(* IEC 61131-3 sources: volt/packages/volt-lsp-iec/test-corpus/CodesysTestProject/Device/Plc Logic/Application/Library Manager/CmpApp, 69 files *)

(* ---- APP_MEMORY_SEGMENT.dut ---- *)
TYPE APP_MEMORY_SEGMENT :
STRUCT
	WTYPE : WORD;
	WAREA : WORD;
	DWOFFSET : DWORD;
	DWSIZE : DWORD;
	DWHIGHESTUSEDADDRESS : DWORD;
END_STRUCT
END_TYPE

(* ---- APPLICATION.dut ---- *)
TYPE APPLICATION :
STRUCT
	PAPPPARENT : POINTER TO APPLICATION;
	IID : UDINT;
	CODEGUID : ARRAY [0..15] OF BYTE;
	DATAGUID : ARRAY [0..15] OF BYTE;
	UDISTATE : UDINT;
	UDIOPSTATE : UDINT;
	HBOOTPROJECT : RTS_IEC_HANDLE;
	HDEBUGTASK : RTS_IEC_HANDLE;
	PFGLOBALINIT : POINTER TO BYTE;
	PFGLOBALEXIT : POINTER TO BYTE;
	HSESSIONIDPOOL : RTS_IEC_HANDLE;
	HFORCEPOOL : RTS_IEC_HANDLE;
	HBPPOOL : RTS_IEC_HANDLE;
	BPERSISTENTFORCE : DINT;
	SZNAME : STRING(MAX_LEN_APPLNAME);
	UDIPSVERSION : UDINT;
	UDITARGETSETTINGVERSION : UDINT;
END_STRUCT
END_TYPE

(* ---- APPLICATION_INFO.dut ---- *)
TYPE APPLICATION_INFO :
STRUCT
	PSTPROJECTNAME : POINTER TO STRING(255);
	PSTAUTHOR : POINTER TO STRING(255);
	PSTVERSION : POINTER TO STRING(255);
	PSTDESCRIPTION : POINTER TO STRING(255);
	PSTPROFILE : POINTER TO STRING(255);
	DTLASTCHANGES : DATE_AND_TIME;
END_STRUCT
END_TYPE

(* ---- EVTPARAM_CMPAPP.dut ---- *)
TYPE EVTPARAM_CMPAPP :
STRUCT
	PAPP : POINTER TO APPLICATION;
END_STRUCT
END_TYPE

(* ---- EVTPARAM_CMPAPPALLBOOTAPPSLOADED.dut ---- *)
TYPE EVTPARAM_CMPAPPALLBOOTAPPSLOADED :
STRUCT
	NTOTALBOOTAPPS : DINT;
	NSUCCESSFULLYLOADEDBOOTAPPS : DINT;
END_STRUCT
END_TYPE

(* ---- EVTPARAM_CMPAPPCOMM.dut ---- *)
TYPE EVTPARAM_CMPAPPCOMM :
STRUCT
	PAPP : POINTER TO APPLICATION;
	UDISESSIONID : UDINT;
	UDIAPPSESSIONID : UDINT;
END_STRUCT
END_TYPE

(* ---- EVTPARAM_CMPAPPCOMMCYCLE.dut ---- *)
TYPE EVTPARAM_CMPAPPCOMMCYCLE :
STRUCT
	ULPARAM1 : __XWORD;
	ULPARAM2 : __XWORD;
END_STRUCT
END_TYPE

(* ---- EVTPARAM_CMPAPPCONFIG.dut ---- *)
TYPE EVTPARAM_CMPAPPCONFIG :
STRUCT
	PAPP : POINTER TO APPLICATION;
	PSZCONFIGAPPLICATION : POINTER TO STRING;
END_STRUCT
END_TYPE

(* ---- EVTPARAM_CMPAPPDELETE.dut ---- *)
TYPE EVTPARAM_CMPAPPDELETE :
STRUCT
	PAPP : POINTER TO APPLICATION;
	ULDELETEREASON : UDINT;
END_STRUCT
END_TYPE

(* ---- EVTPARAM_CMPAPPDENY.dut ---- *)
TYPE EVTPARAM_CMPAPPDENY :
STRUCT
	PAPP : POINTER TO APPLICATION;
	UDIDENY : UDINT;
END_STRUCT
END_TYPE

(* ---- EVTPARAM_CMPAPPDENYDELETE.dut ---- *)
TYPE EVTPARAM_CMPAPPDENYDELETE :
STRUCT
	PAPP : POINTER TO APPLICATION;
	UDISHUTDOWN : UDINT;
	UDIDENY : UDINT;
END_STRUCT
END_TYPE

(* ---- EVTPARAM_CMPAPPDENYLOADBOOTPROJECT.dut ---- *)
TYPE EVTPARAM_CMPAPPDENYLOADBOOTPROJECT :
STRUCT
	PSZAPPNAME : POINTER TO STRING;
	BDENY : DINT;
END_STRUCT
END_TYPE

(* ---- EVTPARAM_CMPAPPDENYSTART.dut ---- *)
TYPE EVTPARAM_CMPAPPDENYSTART :
STRUCT
	PAPP : POINTER TO APPLICATION;
	BDENY : DINT;
END_STRUCT
END_TYPE

(* ---- EVTPARAM_CMPAPPDENYSTOP.dut ---- *)
TYPE EVTPARAM_CMPAPPDENYSTOP :
STRUCT
	PAPP : POINTER TO APPLICATION;
	ULSTOPREASON : DWORD;
	BDENY : DINT;
END_STRUCT
END_TYPE

(* ---- EVTPARAM_CMPAPPEXCEPTION.dut ---- *)
TYPE EVTPARAM_CMPAPPEXCEPTION :
STRUCT
	PAPP : POINTER TO APPLICATION;
	HIECTASK : RTS_IEC_HANDLE;
	UDIEXCEPTION : UDINT;
END_STRUCT
END_TYPE

(* ---- EVTPARAM_CMPAPPEXIT.dut ---- *)
TYPE EVTPARAM_CMPAPPEXIT :
STRUCT
	PAPP : POINTER TO APPLICATION;
	ULEXITREASON : UDINT;
END_STRUCT
END_TYPE

(* ---- EVTPARAM_CMPAPPOEMSERVICETAG.dut ---- *)
TYPE EVTPARAM_CMPAPPOEMSERVICETAG :
STRUCT
	PAPP : POINTER TO APPLICATION;
	UDICHANNELID : UDINT;
	UDITOPLEVELTAG : UDINT;
	UDIHEADERTAG : UDINT;
	UDIREADER : UDINT;
	UDIWRITER : UDINT;
	UDIRESULT : UDINT;
END_STRUCT
END_TYPE

(* ---- EVTPARAM_CMPAPPOPERATINGSTATECHANGED.dut ---- *)
TYPE EVTPARAM_CMPAPPOPERATINGSTATECHANGED :
STRUCT
	PAPP : POINTER TO APPLICATION;
	UDIPREVOPSTATE : UDINT;
END_STRUCT
END_TYPE

(* ---- EVTPARAM_CMPAPPPREPARELOADBOOTPROJECT.dut ---- *)
TYPE EVTPARAM_CMPAPPPREPARELOADBOOTPROJECT :
STRUCT
	PSZAPPNAME : POINTER TO STRING;
END_STRUCT
END_TYPE

(* ---- EVTPARAM_CMPAPPREGISTERBOOTPROJECT.dut ---- *)
TYPE EVTPARAM_CMPAPPREGISTERBOOTPROJECT :
STRUCT
	PSZAPPNAME : POINTER TO STRING;
END_STRUCT
END_TYPE

(* ---- EVTPARAM_CMPAPPRESET.dut ---- *)
TYPE EVTPARAM_CMPAPPRESET :
STRUCT
	PAPP : POINTER TO APPLICATION;
	EWRESETOPTION : RESET_OPTION;
END_STRUCT
END_TYPE

(* ---- EVTPARAM_CMPAPPRESETALLAPPLICATIONS.dut ---- *)
TYPE EVTPARAM_CMPAPPRESETALLAPPLICATIONS :
STRUCT
	EWRESETOPTION : RESET_OPTION;
END_STRUCT
END_TYPE

(* ---- EVTPARAM_CMPAPPRETAINBACKUPSTATE.dut ---- *)
TYPE EVTPARAM_CMPAPPRETAINBACKUPSTATE :
STRUCT
	PSZBOOTPROJECTNAME : POINTER TO STRING;
	UIBACKUPSTATE : UINT;
END_STRUCT
END_TYPE

(* ---- EVTPARAM_CMPAPPSOURCEDOWNLOAD.dut ---- *)
TYPE EVTPARAM_CMPAPPSOURCEDOWNLOAD :
STRUCT
	PSZARCHIVENAME : POINTER TO STRING;
	USIBEGIN : USINT;
END_STRUCT
END_TYPE

(* ---- EVTPARAM_CMPAPPSTATECHANGED.dut ---- *)
TYPE EVTPARAM_CMPAPPSTATECHANGED :
STRUCT
	PAPP : POINTER TO APPLICATION;
	UDIPREVSTATE : UDINT;
END_STRUCT
END_TYPE

(* ---- EVTPARAM_CMPAPPSTOP.dut ---- *)
TYPE EVTPARAM_CMPAPPSTOP :
STRUCT
	PAPP : POINTER TO APPLICATION;
	ULSTOPREASON : DWORD;
END_STRUCT
END_TYPE

(* ---- PROJECT_INFO.dut ---- *)
TYPE PROJECT_INFO :
STRUCT
	STPROJECT : STRING;
	STTITLE : STRING;
	STVERSION : STRING;
	STAUTHOR : STRING;
	STDESCRIPTION : STRING;
END_STRUCT
END_TYPE

(* ---- RESET_OPTION.dut ---- *)
TYPE RESET_OPTION :
(
	RTS_RESET := 0,
	RTS_RESET_COLD := 1,
	RTS_RESET_ORIGIN := 2,
	RTS_RESET_ORIGIN_DEVICE := 3
);
END_TYPE

(* ---- APPLICATIONFLAGS.gvl ---- *)
VAR_GLOBAL
	AF_SYSTEM_APPLICATION : UDINT := 16#10000;
	AF_IOCONFIG_BYTE_ADDRESSING : UDINT := 16#20000;
	AF_IOCONFIG_BIT_WORD_ADDRESSING : UDINT := 16#40000;
	AF_KEEP_AT_PARENT_ONLINE_CHANGE : UDINT := 16#80000;
	AF_ALLOW_SYMBOLIC_VARIABLE_ACCESS_IN_SYNC_WITH_IEC_TASK : UDINT := 16#100000;
	AF_SIGNED_APPLICATION : UDINT := 16#200000;
	AF_ENCRYPTED_APPLICATION : UDINT := 16#400000;
	AF_DEVICE_APPLICATION : UDINT := 16#800000;
	AF_APPLICATION_STOP_PARENT_APPS_ON_EXCEPTION : UDINT := 16#1000000;
END_VAR

(* ---- APPLICATIONSTATE.gvl ---- *)
VAR_GLOBAL
	AS_NONE : UDINT := 16#0;
	AS_RUN : UDINT := 16#1;
	AS_STOP : UDINT := 16#2;
	AS_DEBUG_HALT_ON_BP : UDINT := 16#3;
	AS_DEBUG_STEP : UDINT := 16#4;
	AS_SINGLE_CYCLE : UDINT := 16#5;
END_VAR

(* ---- AREATYPES.gvl ---- *)
VAR_GLOBAL
	DA_NONE : UINT := 16#0;
	DA_DATA : UINT := 16#1;
	DA_CONSTANT : UINT := 16#2;
	DA_INPUT : UINT := 16#4;
	DA_OUTPUT : UINT := 16#8;
	DA_MEMORY : UINT := 16#10;
	DA_RETAIN : UINT := 16#20;
	DA_CODE : UINT := 16#40;
	DA_PERSISTENT : UINT := 16#100;
	DA_ALL : UINT := 16#FFFF;
END_VAR

(* ---- EVENTIDS.gvl ---- *)
VAR_GLOBAL
	CMPID_CMPAPP : DWORD := 16#2;
	EVTPARAMID_CMPAPP : WORD := 16#1;
	EVTVERSION_CMPAPP : WORD := 16#1;
	EVTPARAMID_CMPAPPCONFIG : WORD := 16#1;
	EVTVERSION_CMPAPPCONFIG : WORD := 16#1;
	EVTPARAMID_CMPAPPRESET : WORD := 16#1;
	EVTVERSION_CMPAPPRESET : WORD := 16#2;
	EVTPARAMID_CMPAPPSTOP : WORD := 16#2;
	EVTVERSION_CMPAPPSTOP : WORD := 16#1;
	EVTPARAMID_CMPAPPEXIT : WORD := 16#1;
	EVTVERSION_CMPAPPEXIT : WORD := 16#2;
	EVTPARAMID_CMPAPPDELETE : WORD := 16#1;
	EVTVERSION_CMPAPPDELETE : WORD := 16#2;
	EVTPARAMID_CMPAPPDENYSTART : WORD := 16#3;
	EVTVERSION_CMPAPPDENYSTART : WORD := 16#1;
	EVTPARAMID_CMPAPPDENYSTOP : WORD := 16#4;
	EVTVERSION_CMPAPPDENYSTOP : WORD := 16#1;
	EVTPARAMID_CMPAPPALLBOOTAPPSLOADED : WORD := 16#5;
	EVTVERSION_CMPAPPALLBOOTAPPSLOADED : WORD := 16#1;
	EVTPARAMID_CMPAPPDENYLOADBOOTPROJECT : WORD := 16#6;
	EVTVERSION_CMPAPPDENYLOADBOOTPROJECT : WORD := 16#1;
	EVTPARAMID_CMPAPPPREPARELOADBOOTPROJECT : WORD := 16#7;
	EVTVERSION_CMPAPPPREPARELOADBOOTPROJECT : WORD := 16#1;
	EVTPARAMID_CMPAPPEXCEPTION : WORD := 16#8;
	EVTVERSION_CMPAPPEXCEPTION : WORD := 16#1;
	EVTPARAMID_CMPAPPREGISTERBOOTPROJECT : WORD := 16#9;
	EVTVERSION_CMPAPPREGISTERBOOTPROJECT : WORD := 16#1;
	EVTPARAMID_CMPAPPOPERATINGSTATECHANGED : WORD := 16#A;
	EVTVERSION_CMPAPPOPERATINGSTATECHANGED : WORD := 16#1;
	EVTPARAMID_CMPAPPSOURCEDOWNLOAD : WORD := 16#B;
	EVTVERSION_CMPAPPSOURCEDOWNLOAD : WORD := 16#1;
	EVTPARAMID_CMPAPPCOMM : WORD := 16#C;
	EVTVERSION_CMPAPPCOMM : WORD := 16#2;
	EVTPARAMID_CMPAPPDENY : WORD := 16#D;
	EVTVERSION_CMPAPPDENY : WORD := 16#1;
	EVTPARAMID_CMPAPPDENYDELETE : WORD := 16#E;
	EVTVERSION_CMPAPPDENYDELETE : WORD := 16#1;
	EVTPARAMID_CMPAPPOEMSERVICETAG : WORD := 16#F;
	EVTVERSION_CMPAPPOEMSERVICETAG : WORD := 16#1;
	EVTPARAMID_CMPAPPCOMMCYCLE : WORD := 16#17;
	EVTVERSION_CMPAPPCOMMCYCLE : WORD := 16#1;
	EVTPARAMID_CMPAPPSTATECHANGED : WORD := 16#18;
	EVTVERSION_CMPAPPSTATECHANGED : WORD := 16#1;
	EVTPARAMID_CMPAPPRETAINBACKUPSTATE : WORD := 16#1B;
	EVTVERSION_CMPAPPRETAINBACKUPSTATE : WORD := 16#1;
	EVTPARAMID_CMPAPPRESETALLAPPLICATIONS : WORD := 16#1C;
	EVTVERSION_CMPAPPRESETALLAPPLICATIONS : WORD := 16#1;
	APP_STOP_REASON_UNKNOWN : DWORD := 0;
	APP_STOP_REASON_SHUTDOWN : DWORD := 1;
	APP_STOP_REASON_RESET : DWORD := 2;
	APP_STOP_REASON_EXCEPTION : DWORD := 3;
	APP_STOP_REASON_USER : DWORD := 4;
	APP_STOP_REASON_IECPROGRAM : DWORD := 5;
	APP_STOP_REASON_DELETE : DWORD := 6;
	EVT_PREPARESTART : DWORD := (SHL(UINT_TO_DWORD(EventClass.EVTCLASS_INFO), 16) OR 16#1);
	EVT_STARTDONE : DWORD := (SHL(UINT_TO_DWORD(EventClass.EVTCLASS_INFO), 16) OR 16#2);
	EVT_PREPARESTOP : DWORD := (SHL(UINT_TO_DWORD(EventClass.EVTCLASS_INFO), 16) OR 16#3);
	EVT_STOPDONE : DWORD := (SHL(UINT_TO_DWORD(EventClass.EVTCLASS_INFO), 16) OR 16#4);
	EVT_PREPARERESET : DWORD := (SHL(UINT_TO_DWORD(EventClass.EVTCLASS_INFO), 16) OR 16#5);
	EVT_RESETDONE : DWORD := (SHL(UINT_TO_DWORD(EventClass.EVTCLASS_INFO), 16) OR 16#6);
	EVT_PREPAREONLINECHANGE : DWORD := (SHL(UINT_TO_DWORD(EventClass.EVTCLASS_INFO), 16) OR 16#7);
	EVT_ONLINECHANGEDONE : DWORD := (SHL(UINT_TO_DWORD(EventClass.EVTCLASS_INFO), 16) OR 16#8);
	EVT_PREPAREDOWNLOAD : DWORD := (SHL(UINT_TO_DWORD(EventClass.EVTCLASS_INFO), 16) OR 16#9);
	EVT_DOWNLOADDONE : DWORD := (SHL(UINT_TO_DWORD(EventClass.EVTCLASS_INFO), 16) OR 16#A);
	EVT_CODEINITDONE : DWORD := (SHL(UINT_TO_DWORD(EventClass.EVTCLASS_INFO), 16) OR 16#B);
	EVT_PREPAREDELETE : DWORD := (SHL(UINT_TO_DWORD(EventClass.EVTCLASS_INFO), 16) OR 16#C);
	EVT_DELETEDONE : DWORD := (SHL(UINT_TO_DWORD(EventClass.EVTCLASS_INFO), 16) OR 16#D);
	EVT_PREPAREEXIT : DWORD := (SHL(UINT_TO_DWORD(EventClass.EVTCLASS_INFO), 16) OR 16#E);
	EVT_EXITDONE : DWORD := (SHL(UINT_TO_DWORD(EventClass.EVTCLASS_INFO), 16) OR 16#F);
	EVT_CREATEBOOTPROJECTDONE : DWORD := (SHL(UINT_TO_DWORD(EventClass.EVTCLASS_INFO), 16) OR 16#10);
	EVT_DENYLOADBOOTPROJECT : DWORD := (SHL(UINT_TO_DWORD(EventClass.EVTCLASS_INFO), 16) OR 16#12);
	EVT_PREPARELOADBOOTPROJECT : DWORD := (SHL(UINT_TO_DWORD(EventClass.EVTCLASS_INFO), 16) OR 16#13);
	EVT_LOADBOOTPROJECTDONE : DWORD := (SHL(UINT_TO_DWORD(EventClass.EVTCLASS_INFO), 16) OR 16#11);
	EVT_DENYSTARTBOOTPROJECT : DWORD := (SHL(UINT_TO_DWORD(EventClass.EVTCLASS_INFO), 16) OR 16#14);
	EVT_PREPARESTARTBOOTPROJECT : DWORD := (SHL(UINT_TO_DWORD(EventClass.EVTCLASS_INFO), 16) OR 16#15);
	EVT_STARTBOOTPROJECTDONE : DWORD := (SHL(UINT_TO_DWORD(EventClass.EVTCLASS_INFO), 16) OR 16#16);
	EVT_DENYSTART : DWORD := (SHL(UINT_TO_DWORD(EventClass.EVTCLASS_INFO), 16) OR 16#17);
	EVT_DENYSTOP : DWORD := (SHL(UINT_TO_DWORD(EventClass.EVTCLASS_INFO), 16) OR 16#18);
	EVT_ALLBOOTPROJECTSLOADED : DWORD := (SHL(UINT_TO_DWORD(EventClass.EVTCLASS_INFO), 16) OR 16#19);
	EVT_GLOBALEXITONRESETDONE : DWORD := (SHL(UINT_TO_DWORD(EventClass.EVTCLASS_INFO), 16) OR 16#1A);
	EVT_EXITDONEWITHCONFIGAPPINFO : DWORD := (SHL(UINT_TO_DWORD(EventClass.EVTCLASS_INFO), 16) OR 16#1B);
	EVT_CMPAPP_EXCEPTION : DWORD := (SHL(UINT_TO_DWORD(EventClass.EVTCLASS_EXCEPTION), 16) OR 16#1C);
	EVT_REGISTERBOOTPROJECT : DWORD := (SHL(UINT_TO_DWORD(EventClass.EVTCLASS_INFO), 16) OR 16#1D);
	EVT_CREATEBOOTPROJECTFILEFAILED : DWORD := (SHL(UINT_TO_DWORD(EventClass.EVTCLASS_ERROR), 16) OR 16#1E);
	EVT_CREATEBOOTPROJECTFAILED : DWORD := (SHL(UINT_TO_DWORD(EventClass.EVTCLASS_ERROR), 16) OR 16#1F);
	EVT_OPERATINGSTATECHANGED : DWORD := (SHL(UINT_TO_DWORD(EventClass.EVTCLASS_INFO), 16) OR 16#20);
	EVT_OPERATIONSTATECHANGED : DWORD := (SHL(UINT_TO_DWORD(EventClass.EVTCLASS_INFO), 16) OR 16#20);
	EVT_SOURCEDOWNLOAD : DWORD := (SHL(UINT_TO_DWORD(EventClass.EVTCLASS_INFO), 16) OR 16#21);
	EVT_LOGIN : DWORD := (SHL(UINT_TO_DWORD(EventClass.EVTCLASS_INFO), 16) OR 16#22);
	EVT_LOGOUT : DWORD := (SHL(UINT_TO_DWORD(EventClass.EVTCLASS_INFO), 16) OR 16#23);
	EVT_DENYDELETE : DWORD := (SHL(UINT_TO_DWORD(EventClass.EVTCLASS_INFO), 16) OR 16#24);
	EVT_DENYDELETEBOOTPROJECT : DWORD := (SHL(UINT_TO_DWORD(EventClass.EVTCLASS_INFO), 16) OR 16#25);
	EVT_OEMDOWNLOADSERVICETAG : DWORD := (SHL(UINT_TO_DWORD(EventClass.EVTCLASS_INFO), 16) OR 16#27);
	EVT_COMMCYCLE : DWORD := (SHL(UINT_TO_DWORD(EventClass.EVTCLASS_INFO), 16) OR 16#2A);
	EVT_STATECHANGED : DWORD := (SHL(UINT_TO_DWORD(EventClass.EVTCLASS_INFO), 16) OR 16#2B);
	EVT_RETAINBACKUPSTATE : DWORD := (SHL(UINT_TO_DWORD(EventClass.EVTCLASS_INFO), 16) OR 16#2F);
	EVT_RESETALLAPPLICATIONS_PREPARE : DWORD := (SHL(UINT_TO_DWORD(EventClass.EVTCLASS_INFO), 16) OR 16#30);
	EVT_RESETALLAPPLICATIONS_DONE : DWORD := (SHL(UINT_TO_DWORD(EventClass.EVTCLASS_INFO), 16) OR 16#31);
END_VAR

(* ---- EXCEPTION.gvl ---- *)
VAR_GLOBAL
	RTSEXCPT_APP_TARGET_MISMATCH : DWORD := 16#26;
END_VAR

(* ---- GLOBALCONSTANTS.gvl ---- *)
VAR_GLOBAL
	MAX_LEN_APPLNAME : UDINT := 60;
END_VAR

(* ---- OPERATINGSTATE.gvl ---- *)
VAR_GLOBAL
	OS_NONE : UDINT := 16#0;
	OS_PROGRAM_LOADED : UDINT := 16#1;
	OS_DOWNLOAD : UDINT := 16#2;
	OS_ONLINE_CHANGE : UDINT := 16#4;
	OS_STORE_BOOTPROJECT : UDINT := 16#8;
	OS_FORCE_ACTIVE : UDINT := 16#10;
	OS_EXCEPTION : UDINT := 16#20;
	OS_RUN_AFTER_DOWNLOAD : UDINT := 16#40;
	OS_STORE_BOOTPROJECT_ONLY : UDINT := 16#80;
END_VAR

(* ---- OPERATIONREASON.gvl ---- *)
VAR_GLOBAL
	APP_REASON_UNKNOWN : UDINT := 16#0;
	APP_REASON_SHUTDOWN : UDINT := 16#1;
	APP_REASON_RESET : UDINT := 16#2;
	APP_REASON_EXCEPTION : UDINT := 16#3;
	APP_REASON_USER : UDINT := 16#4;
	APP_REASON_IECPROGRAM : UDINT := 16#5;
	APP_REASON_DELETE : UDINT := 16#6;
	APP_REASON_DEBUGGING : UDINT := 16#7;
	APP_REASON_RUNSTOP_SWITCH : UDINT := 16#8;
	APP_REASON_REDUNDANCY_SYNC : UDINT := 16#9;
END_VAR

(* ---- OPERATIONS.gvl ---- *)
VAR_GLOBAL
	OP_APP_STOP : UDINT := 1;
	OP_APP_DOWNLOAD : UDINT := 2;
	OP_APP_ONLINECHANGE : UDINT := 3;
	OP_APP_WRITE_VARIABLES : UDINT := 4;
	OP_APP_FORCE_VARIABLES : UDINT := 5;
	OP_APP_SET_BREAKPOINT : UDINT := 6;
	OP_APP_RESET : UDINT := 7;
	OP_APP_START : UDINT := 8;
	OP_APP_DELETE_APPLICATION : UDINT := 9;
	OP_APP_RESET_ORIGIN : UDINT := 10;
END_VAR

(* ---- RETAINBACKUPSTATE.gvl ---- *)
VAR_GLOBAL
	APP_RBS_UNKNOWN : UINT := 0;
	APP_RBS_BACKUP_PREPARE : UINT := 1;
	APP_RBS_BACKUP_BEGIN : UINT := 2;
	APP_RBS_BACKUP_END : UINT := 3;
	APP_RBS_RESTORE : UINT := 4;
END_VAR

(* ---- APPCALLGETPROPERTY.pou ---- *)
FUNCTION APPCALLGETPROPERTY : RTS_IEC_RESULT
VAR_INPUT
	PINSTANCE : POINTER TO BYTE;
	PPGETMETHOD : POINTER TO POINTER TO BYTE;
	PBYVALUE : POINTER TO BYTE;
	ULSIZE : __XWORD;
END_VAR
END_FUNCTION

(* ---- APPCALLGETPROPERTY2.pou ---- *)
FUNCTION APPCALLGETPROPERTY2 : RTS_IEC_RESULT
VAR_INPUT
	PINSTANCE : POINTER TO BYTE;
	PPGETMETHOD : POINTER TO POINTER TO BYTE;
	PPBYVALUE : POINTER TO POINTER TO BYTE;
	ULSIZE : __XWORD;
END_VAR
END_FUNCTION

(* ---- APPCALLGETPROPERTY2RELEASE.pou ---- *)
FUNCTION APPCALLGETPROPERTY2RELEASE : RTS_IEC_RESULT
VAR_INPUT
	PBYVALUE : POINTER TO BYTE;
END_VAR
END_FUNCTION

(* ---- APPCALLGETPROPERTY3.pou ---- *)
FUNCTION APPCALLGETPROPERTY3 : RTS_IEC_RESULT
VAR_INPUT
	PINSTANCE : POINTER TO BYTE;
	PPGETMETHOD : POINTER TO POINTER TO BYTE;
	PPBYVALUE : POINTER TO POINTER TO BYTE;
	ULSIZE : __XWORD;
	ULOFFSET : __XWORD;
END_VAR
END_FUNCTION

(* ---- APPCALLSETPROPERTY.pou ---- *)
FUNCTION APPCALLSETPROPERTY : RTS_IEC_RESULT
VAR_INPUT
	PINSTANCE : POINTER TO BYTE;
	PPSETMETHOD : POINTER TO POINTER TO BYTE;
	PBYVALUE : POINTER TO BYTE;
	ULSIZE : __XWORD;
END_VAR
END_FUNCTION

(* ---- APPCALLSETPROPERTY2.pou ---- *)
FUNCTION APPCALLSETPROPERTY2 : RTS_IEC_RESULT
VAR_INPUT
	PINSTANCE : POINTER TO BYTE;
	PPSETMETHOD : POINTER TO POINTER TO BYTE;
	PBYVALUE : POINTER TO BYTE;
	ULSIZE : __XWORD;
	ULOFFSET : __XWORD;
END_VAR
END_FUNCTION

(* ---- APPCHECKBOOTPROJECTCONSISTENCY.pou ---- *)
FUNCTION APPCHECKBOOTPROJECTCONSISTENCY : RTS_IEC_RESULT
VAR_INPUT
	PAPP : POINTER TO APPLICATION;
END_VAR
END_FUNCTION

(* ---- APPFINDAPPLICATIONBYNAME.pou ---- *)
FUNCTION APPFINDAPPLICATIONBYNAME : POINTER TO APPLICATION
VAR_INPUT
	PSZSTRING : REFERENCE TO STRING;
	PRESULT : POINTER TO RTS_IEC_RESULT;
END_VAR
END_FUNCTION

(* ---- APPGENERATEEXCEPTION.pou ---- *)
FUNCTION APPGENERATEEXCEPTION : RTS_IEC_RESULT
VAR_INPUT
	PAPP : POINTER TO APPLICATION;
	ULEXCEPTION : DWORD;
END_VAR
END_FUNCTION

(* ---- APPGETAPPLICATIONBYAREAADDRESS.pou ---- *)
FUNCTION APPGETAPPLICATIONBYAREAADDRESS : POINTER TO APPLICATION
VAR_INPUT
	PADDRESS : POINTER TO UDINT;
END_VAR
END_FUNCTION

(* ---- APPGETAPPLICATIONFLAGS.pou ---- *)
FUNCTION APPGETAPPLICATIONFLAGS : UDINT
VAR_INPUT
	PAPP : POINTER TO APPLICATION;
	PRESULT : POINTER TO RTS_IEC_RESULT;
END_VAR
END_FUNCTION

(* ---- APPGETAPPLICATIONINFO.pou ---- *)
FUNCTION APPGETAPPLICATIONINFO : POINTER TO APPLICATION_INFO
VAR_INPUT
	PAPP : POINTER TO APPLICATION;
	PRESULT : POINTER TO RTS_IEC_RESULT;
END_VAR
END_FUNCTION

(* ---- APPGETAREAADDRESS.pou ---- *)
FUNCTION APPGETAREAADDRESS : POINTER TO BYTE
VAR_INPUT
	PAPP : POINTER TO APPLICATION;
	UITYPE : UINT;
	PRESULT : POINTER TO RTS_IEC_RESULT;
END_VAR
END_FUNCTION

(* ---- APPGETAREAOFFSETBYADDRESS.pou ---- *)
FUNCTION APPGETAREAOFFSETBYADDRESS : RTS_IEC_RESULT
VAR_INPUT
	PAPP : POINTER TO APPLICATION;
	ULADDRESS : __UXINT;
	PUSAREA : POINTER TO WORD;
	PULOFFSET : POINTER TO __XWORD;
END_VAR
END_FUNCTION

(* ---- APPGETAREAPOINTER.pou ---- *)
FUNCTION APPGETAREAPOINTER : RTS_IEC_RESULT
VAR_INPUT
	PAPP : POINTER TO APPLICATION;
	DIAREA : DINT;
	PPBYAREA : POINTER TO POINTER TO BYTE;
END_VAR
END_FUNCTION

(* ---- APPGETAREASIZE.pou ---- *)
FUNCTION APPGETAREASIZE : __XWORD
VAR_INPUT
	PAPP : POINTER TO APPLICATION;
	UITYPE : UINT;
	PRESULT : POINTER TO RTS_IEC_RESULT;
END_VAR
END_FUNCTION

(* ---- APPGETCURRENT.pou ---- *)
FUNCTION APPGETCURRENT : POINTER TO APPLICATION
VAR_INPUT
	PRESULT : POINTER TO RTS_IEC_RESULT;
END_VAR
END_FUNCTION

(* ---- APPGETFIRSTAPP.pou ---- *)
FUNCTION APPGETFIRSTAPP : POINTER TO APPLICATION
VAR_INPUT
	PRESULT : POINTER TO RTS_IEC_RESULT;
END_VAR
END_FUNCTION

(* ---- APPGETNEXTAPP.pou ---- *)
FUNCTION APPGETNEXTAPP : POINTER TO APPLICATION
VAR_INPUT
	PAPPPREV : POINTER TO APPLICATION;
	PRESULT : POINTER TO RTS_IEC_RESULT;
END_VAR
END_FUNCTION

(* ---- APPGETPROJECTINFORMATION.pou ---- *)
FUNCTION APPGETPROJECTINFORMATION : RTS_IEC_RESULT
VAR_INPUT
	PAPP : POINTER TO APPLICATION;
	PINFO : POINTER TO PROJECT_INFO;
END_VAR
END_FUNCTION

(* ---- APPGETSEGMENT.pou ---- *)
FUNCTION APPGETSEGMENT : POINTER TO APP_MEMORY_SEGMENT
VAR_INPUT
	PAPP : POINTER TO APPLICATION;
	UITYPE : UINT;
	PRESULT : POINTER TO RTS_IEC_RESULT;
END_VAR
END_FUNCTION

(* ---- APPGETSEGMENTADDRESS.pou ---- *)
FUNCTION APPGETSEGMENTADDRESS : POINTER TO BYTE
VAR_INPUT
	PAPP : POINTER TO APPLICATION;
	WTYPE : WORD;
	PRESULT : POINTER TO RTS_IEC_RESULT;
END_VAR
END_FUNCTION

(* ---- APPGETSEGMENTSIZE.pou ---- *)
FUNCTION APPGETSEGMENTSIZE : __UXINT
VAR_INPUT
	PAPP : POINTER TO APPLICATION;
	WTYPE : WORD;
	PRESULT : POINTER TO RTS_IEC_RESULT;
END_VAR
END_FUNCTION

(* ---- APPNUMOFACTIVESESSIONS.pou ---- *)
FUNCTION APPNUMOFACTIVESESSIONS : RTS_IEC_RESULT
VAR_INPUT
	PAPP : POINTER TO APPLICATION;
	PULNUMSESSIONS : POINTER TO UDINT;
END_VAR
END_FUNCTION

(* ---- APPREGISTERPROPACCESSFUNCTIONS.pou ---- *)
FUNCTION APPREGISTERPROPACCESSFUNCTIONS : RTS_IEC_RESULT
VAR_INPUT
	PAPP : POINTER TO APPLICATION;
	PPFGETBOOLEANPROPERTY : POINTER TO POINTER TO BYTE;
	PPFGETTEXTPROPERTY : POINTER TO POINTER TO BYTE;
	PPFGETNUMBERPROPERTY : POINTER TO POINTER TO BYTE;
	PPFGETVERSIONPROPERTY : POINTER TO POINTER TO BYTE;
END_VAR
END_FUNCTION

(* ---- APPRESET.pou ---- *)
FUNCTION APPRESET : RTS_IEC_RESULT
VAR_INPUT
	PAPP : POINTER TO APPLICATION;
	USRESETOPTION : WORD;
END_VAR
END_FUNCTION

(* ---- APPRESTORERETAINSFROMFILE.pou ---- *)
FUNCTION APPRESTORERETAINSFROMFILE : RTS_IEC_RESULT
VAR_INPUT
	PAPP : POINTER TO APPLICATION;
	PSZFILNAME : REFERENCE TO STRING;
END_VAR
END_FUNCTION

(* ---- APPSTARTAPPLICATION.pou ---- *)
FUNCTION APPSTARTAPPLICATION : RTS_IEC_RESULT
VAR_INPUT
	PAPP : POINTER TO APPLICATION;
END_VAR
END_FUNCTION

(* ---- APPSTOPAPPLICATION.pou ---- *)
FUNCTION APPSTOPAPPLICATION : RTS_IEC_RESULT
VAR_INPUT
	PAPP : POINTER TO APPLICATION;
END_VAR
END_FUNCTION

(* ---- APPSTORERETAINSINFILE.pou ---- *)
FUNCTION APPSTORERETAINSINFILE : RTS_IEC_RESULT
VAR_INPUT
	PAPP : POINTER TO APPLICATION;
	PSZFILNAME : REFERENCE TO STRING;
END_VAR
END_FUNCTION

(* ---- MAKE_EVENTID.pou ---- *)
FUNCTION MAKE_EVENTID : DWORD
VAR_INPUT
	CLASS : UINT;
	EVENTID : UINT;
END_VAR
END_FUNCTION
